// TIA Portal V19 export
FUNCTION_BLOCK "FDevice_Valve_FB"   // FB57, F_LAD
TITLE = FDevice Valve Safety Cutoff + Ev Degas
// stored: Access Published
   VAR_INPUT
      C_FEEDBACK : Bool;   // Contactor feedback
      V_FEEDBACK_CHA : Bool;   // Safety Valve Feedback Channel A
      V_FEEDBACK_CHB : Bool;   // Safety Valve Feedback Channel B
      DEGAS_FEEDBACK : Bool;   // Degas Valve Feedback
      QBAD_FIO : Bool;   // Safety valve Output QBAD_FIO
      Estop : Bool;
      Two_Hand_CMD : Bool;   // Safe Motion Command
      Door_SafeStop : Bool;   // Safe Stop from Doors
      CtrlSafe : Bool;   // Movement is Required
      Reset : Bool;
      StoppingTime : Time := T#2S;   // Movement stopping time
      EvDegasExist : Bool;   // Degas valve Exist
      EvDegasTime : Time := T#500MS;   // Delay On Ev degas after Ev Safety
      SafeStateTime : Time := T#5S;   // Delay for device safe state if V Feedback don't work
   END_VAR
   VAR_OUTPUT
      EV_SAFETY : Bool;   // EV Safety cutoff output
      EV_DEGAS : Bool;   // EV Degas output
      FDO_FBK_ERROR : Bool;   // FDO Feedback error (QBAD Feedback error)
      EV_SAFETY_FBK_WARNING : Bool;   // Ev Safety feedback warning
      EV_DEGAS_FBK_WARNING : Bool;   // Ev Degas feedback warning
   END_VAR
   VAR_IN_OUT
      DSI : "udt_DeviceSafetyInterface";   // Device Safety Interface
   END_VAR
   VAR
      EV_FDBACK : FDBACK;
      T_StopDelay : TOF;
      T_SafeState { S7_SetPoint := 'True'} : TON;
      T_EvSafetyFbk : TON;
      T_EvDegas : TON;
      T_EvDegasFbk : TON;
   END_VAR
   VAR_TEMP
      S_ON : Bool;
   END_VAR
BEGIN

REGION Network 1: Safety Enable
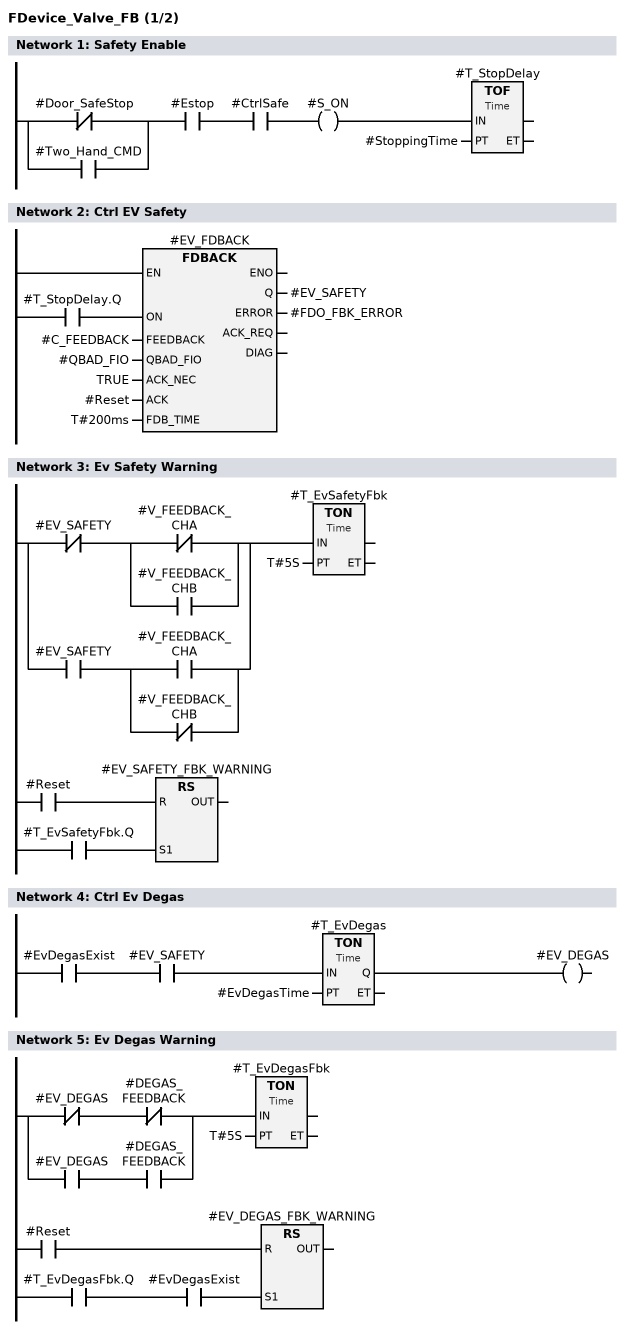
   RUNG wire#powerrail
      I_Contact( #Door_SafeStop )
      wire#w1
      Contact( #Estop )
      Contact( #CtrlSafe )
      Coil( #S_ON )
      { S7_Templates := "[time_type := Time, codedbool_type := DInt]" } #T_StopDelay.TOF(pt := #StoppingTime, et =>)
   END_RUNG
   RUNG wire#powerrail
      Contact( #Two_Hand_CMD )
   END_RUNG wire#w1
   // the same network as SCL:
   #S_ON := (NOT #Door_SafeStop OR #Two_Hand_CMD) AND #Estop AND #CtrlSafe;
   #T_StopDelay.TOF(IN := #S_ON, PT := #StoppingTime);
END_REGION

REGION Network 2: Ctrl EV Safety
   RUNG wire#powerrail
      #EV_FDBACK.FDBACK(ON := wire#w1, FEEDBACK := #C_FEEDBACK, QBAD_FIO := #QBAD_FIO, ACK_NEC := TRUE, ACK := #Reset, FDB_TIME := T#200ms, Q => #EV_SAFETY, ERROR => #FDO_FBK_ERROR, ACK_REQ =>, DIAG =>)
   END_RUNG
   RUNG wire#powerrail
      Contact( #T_StopDelay.Q )
   END_RUNG wire#w1
   // the same network as SCL:
   #EV_FDBACK(ON := #T_StopDelay.Q,   // FDBACK
              FEEDBACK := #C_FEEDBACK,
              QBAD_FIO := #QBAD_FIO,
              ACK_NEC := TRUE,
              ACK := #Reset,
              FDB_TIME := T#200ms,
              Q => #EV_SAFETY,
              ERROR => #FDO_FBK_ERROR);
END_REGION

REGION Network 3: Ev Safety Warning
   RUNG wire#powerrail
      I_Contact( #EV_SAFETY )
      wire#w1
      I_Contact( #V_FEEDBACK_CHA )
      wire#w2
      { S7_Templates := "[time_type := Time, codedbool_type := DInt]" } #T_EvSafetyFbk.TON(pt := T#5S, et =>)
   END_RUNG
   RUNG wire#w1
      Contact( #V_FEEDBACK_CHB )
   END_RUNG wire#w2
   RUNG wire#powerrail
      Contact( #EV_SAFETY )
      wire#w3
      Contact( #V_FEEDBACK_CHA )
   END_RUNG wire#w2
   RUNG wire#w3
      I_Contact( #V_FEEDBACK_CHB )
   END_RUNG wire#w2
   RUNG wire#powerrail
      Contact( #Reset )
      S_RS(operand := #EV_SAFETY_FBK_WARNING, s1 := wire#w4)
   END_RUNG
   RUNG wire#powerrail
      Contact( #T_EvSafetyFbk.Q )
   END_RUNG wire#w4
   // the same network as SCL:
   #T_EvSafetyFbk.TON(IN := (NOT #EV_SAFETY AND (NOT #V_FEEDBACK_CHA OR #V_FEEDBACK_CHB)) OR (#EV_SAFETY AND (#V_FEEDBACK_CHA OR NOT #V_FEEDBACK_CHB)),
                      PT := T#5S);
   IF #Reset THEN
       #EV_SAFETY_FBK_WARNING := FALSE;   // RS flip-flop
   END_IF;
   IF #T_EvSafetyFbk.Q THEN #EV_SAFETY_FBK_WARNING := TRUE; END_IF;
END_REGION

REGION Network 4: Ctrl Ev Degas
   RUNG wire#powerrail
      Contact( #EvDegasExist )
      Contact( #EV_SAFETY )
      { S7_Templates := "[time_type := Time, codedbool_type := DInt]" } #T_EvDegas.TON(pt := #EvDegasTime, et =>)
      Coil( #EV_DEGAS )
   END_RUNG
   // the same network as SCL:
   #T_EvDegas.TON(IN := #EvDegasExist AND #EV_SAFETY, PT := #EvDegasTime);
   #EV_DEGAS := #T_EvDegas.Q;
END_REGION

REGION Network 5: Ev Degas Warning
   RUNG wire#powerrail
      I_Contact( #EV_DEGAS )
      I_Contact( #DEGAS_FEEDBACK )
      wire#w1
      { S7_Templates := "[time_type := Time, codedbool_type := DInt]" } #T_EvDegasFbk.TON(pt := T#5S, et =>)
   END_RUNG
   RUNG wire#powerrail
      Contact( #EV_DEGAS )
      Contact( #DEGAS_FEEDBACK )
   END_RUNG wire#w1
   RUNG wire#powerrail
      Contact( #Reset )
      S_RS(operand := #EV_DEGAS_FBK_WARNING, s1 := wire#w2)
   END_RUNG
   RUNG wire#powerrail
      Contact( #T_EvDegasFbk.Q )
      Contact( #EvDegasExist )
   END_RUNG wire#w2
   // the same network as SCL:
   #T_EvDegasFbk.TON(IN := (NOT #EV_DEGAS AND NOT #DEGAS_FEEDBACK) OR (#EV_DEGAS AND #DEGAS_FEEDBACK),
                     PT := T#5S);
   IF #Reset THEN
       #EV_DEGAS_FBK_WARNING := FALSE;   // RS flip-flop
   END_IF;
   IF #T_EvDegasFbk.Q AND #EvDegasExist THEN #EV_DEGAS_FBK_WARNING := TRUE; END_IF;
END_REGION

REGION Network 6: Enable Power
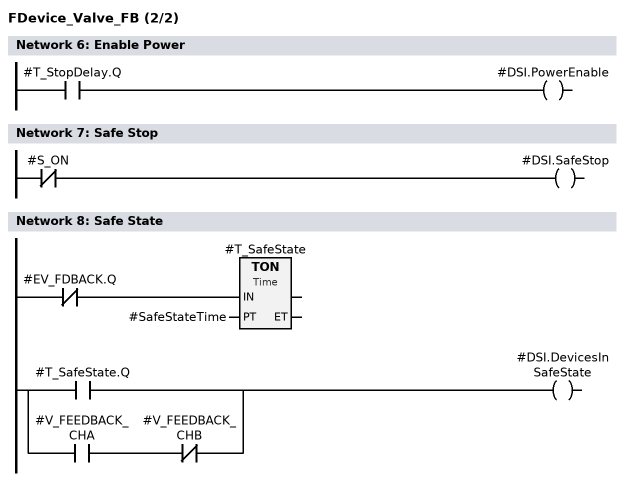
   RUNG wire#powerrail
      Contact( #T_StopDelay.Q )
      Coil( #DSI.PowerEnable )
   END_RUNG
   // the same network as SCL:
   #DSI.PowerEnable := #T_StopDelay.Q;
END_REGION

REGION Network 7: Safe Stop
   RUNG wire#powerrail
      I_Contact( #S_ON )
      Coil( #DSI.SafeStop )
   END_RUNG
   // the same network as SCL:
   #DSI.SafeStop := NOT #S_ON;
END_REGION

REGION Network 8: Safe State
   RUNG wire#powerrail
      I_Contact( #EV_FDBACK.Q )
      { S7_Templates := "[time_type := Time, codedbool_type := DInt]" } #T_SafeState.TON(pt := #SafeStateTime, et =>)
   END_RUNG
   RUNG wire#powerrail
      Contact( #T_SafeState.Q )
      wire#w1
      Coil( #DSI.DevicesInSafeState )
   END_RUNG
   RUNG wire#powerrail
      Contact( #V_FEEDBACK_CHA )
      I_Contact( #V_FEEDBACK_CHB )
   END_RUNG wire#w1
   // the same network as SCL:
   #T_SafeState.TON(IN := NOT #EV_FDBACK.Q, PT := #SafeStateTime);
   #DSI.DevicesInSafeState := #T_SafeState.Q OR (#V_FEEDBACK_CHA AND NOT #V_FEEDBACK_CHB);
END_REGION
END_FUNCTION_BLOCK
